GLOBALCONSTANTS isobus (* Global constants *)
  (* Standard: 61499-1; Description: Copyright (c) 2023 franz This program and the accompanying materials are made available under the terms of the Eclipse Public License 2.0 which is available at https://www.eclipse.org/legal/epl-2.0/ SPDX-License-Identifier: EPL-2.0 *)
  (* Version 1.0, 2023-10-22, franz *)
  VAR_GLOBAL CONSTANT
    ID_NULL : UINT := UINT#16#FFFF;
    ID_OFF : UINT := UINT#16#0;
    GLOBAL : USINT := USINT#16#FF;
    OFF : USINT := USINT#16#0;
  END_VAR
END_GLOBALCONSTANTS
